TYPE EL6001_COM_Outputs :
STRUCT
	{attribute addProperty Name "Control"}
	Control AT %Q* : EL6001_Control;
	{attribute addProperty Name "Data"}
	Data  AT %Q* : ARRAY[0..21] OF USINT;
END_STRUCT
END_TYPE

(* stored: Version 1.1.0.1, ProductVersion 3.1.4024.9
   DUT EL6001_COM_Outputs: Id {27a8c148-2180-0ac9-1da1-18193525313b} *)
